// Mitsubishi GX Works2 project: 增压   PLC: FX1S

PROGRAM MAIN
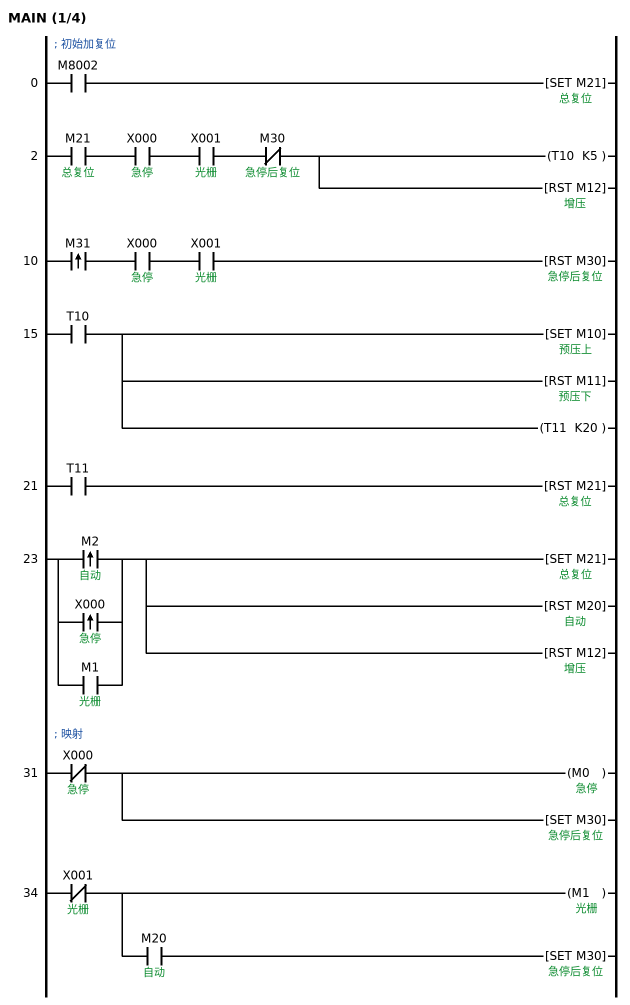
; 初始加复位
0     LD      M8002
      SET     M21  ; 总复位
2     LD      M21  ; 总复位
      AND     X000  ; 急停
      AND     X001  ; 光栅
      ANI     M30  ; 急停后复位
      OUT     T10 K5
      RST     M12  ; 增压
10    LDP     M31
      AND     X000  ; 急停
      AND     X001  ; 光栅
      RST     M30  ; 急停后复位
15    LD      T10
      SET     M10  ; 预压上
      RST     M11  ; 预压下
      OUT     T11 K20
21    LD      T11
      RST     M21  ; 总复位
23    LDP     M2  ; 自动
      ORP     X000  ; 急停
      OR      M1  ; 光栅
      SET     M21  ; 总复位
      RST     M20  ; 自动
      RST     M12  ; 增压
; 映射
31    LDI     X000  ; 急停
      OUT     M0  ; 急停
      SET     M30  ; 急停后复位
34    LDI     X001  ; 光栅
      OUT     M1  ; 光栅
      AND     M20  ; 自动
      SET     M30  ; 急停后复位
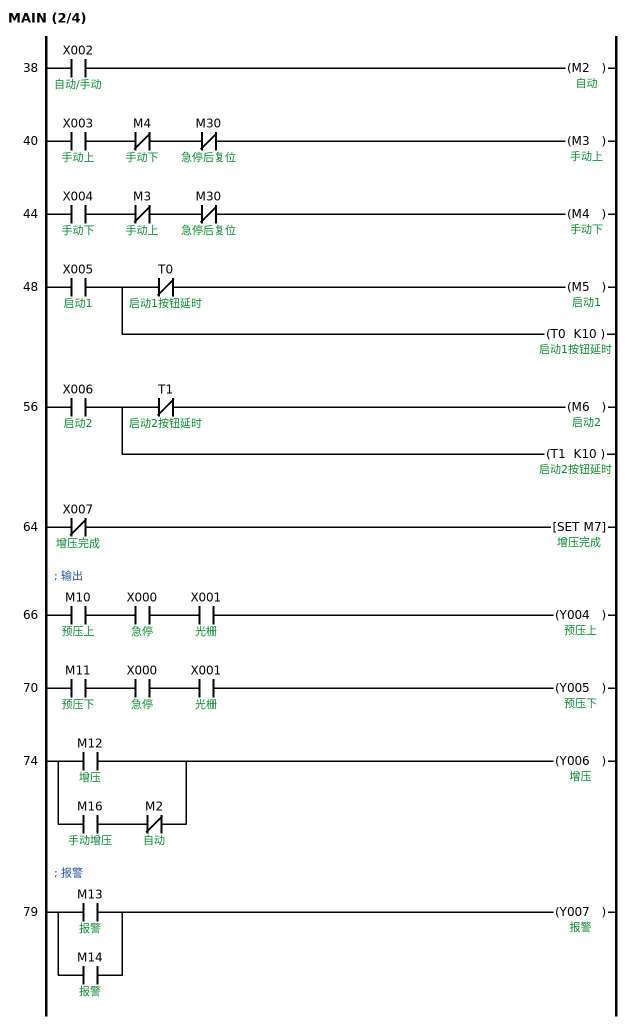
38    LD      X002  ; 自动/手动
      OUT     M2  ; 自动
40    LD      X003  ; 手动上
      ANI     M4  ; 手动下
      ANI     M30  ; 急停后复位
      OUT     M3  ; 手动上
44    LD      X004  ; 手动下
      ANI     M3  ; 手动上
      ANI     M30  ; 急停后复位
      OUT     M4  ; 手动下
48    LD      X005  ; 启动1
      MPS
      ANI     T0  ; 启动1按钮延时
      OUT     M5  ; 启动1
      MPP
      OUT     T0 K10  ; 启动1按钮延时
56    LD      X006  ; 启动2
      MPS
      ANI     T1  ; 启动2按钮延时
      OUT     M6  ; 启动2
      MPP
      OUT     T1 K10  ; 启动2按钮延时
64    LDI     X007  ; 增压完成
      SET     M7  ; 增压完成
; 输出
66    LD      M10  ; 预压上
      AND     X000  ; 急停
      AND     X001  ; 光栅
      OUT     Y004  ; 预压上
70    LD      M11  ; 预压下
      AND     X000  ; 急停
      AND     X001  ; 光栅
      OUT     Y005  ; 预压下
74    LD      M12  ; 增压
      LD      M16  ; 手动增压
      ANI     M2  ; 自动
      ORB
      OUT     Y006  ; 增压
; 报警
79    LD      M13  ; 报警
      OR      M14  ; 报警
      OUT     Y007  ; 报警
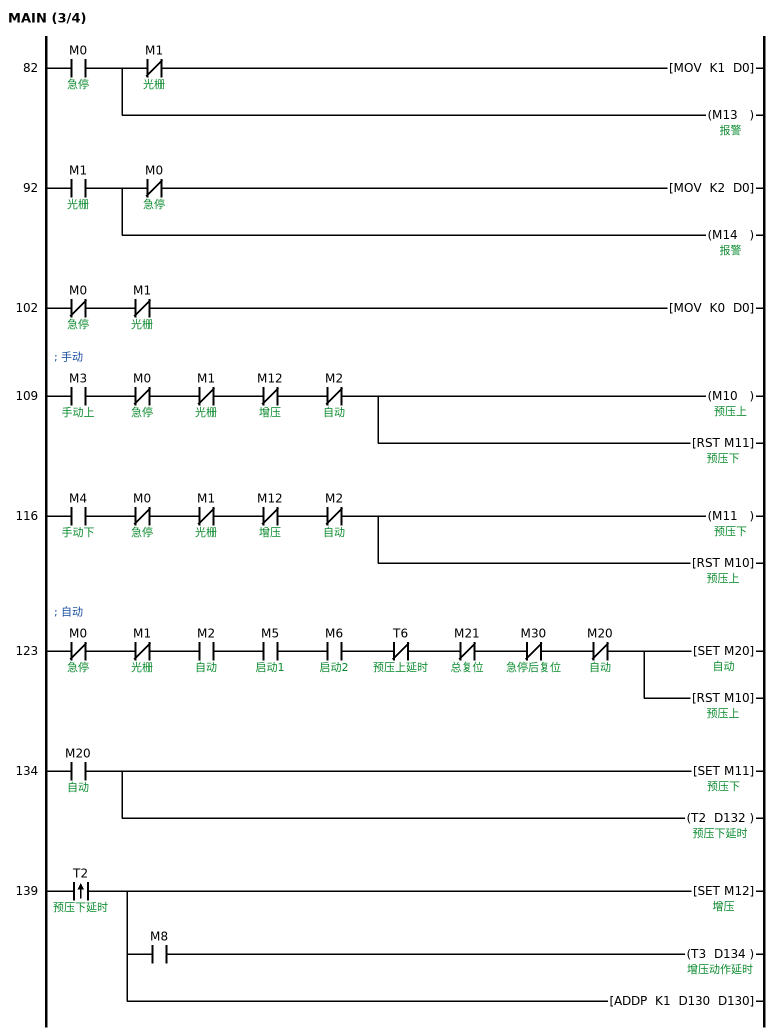
82    LD      M0  ; 急停
      MPS
      ANI     M1  ; 光栅
      MOV     K1 D0
      MPP
      OUT     M13  ; 报警
92    LD      M1  ; 光栅
      MPS
      ANI     M0  ; 急停
      MOV     K2 D0
      MPP
      OUT     M14  ; 报警
102   LDI     M0  ; 急停
      ANI     M1  ; 光栅
      MOV     K0 D0
; 手动
109   LD      M3  ; 手动上
      ANI     M0  ; 急停
      ANI     M1  ; 光栅
      ANI     M12  ; 增压
      ANI     M2  ; 自动
      OUT     M10  ; 预压上
      RST     M11  ; 预压下
116   LD      M4  ; 手动下
      ANI     M0  ; 急停
      ANI     M1  ; 光栅
      ANI     M12  ; 增压
      ANI     M2  ; 自动
      OUT     M11  ; 预压下
      RST     M10  ; 预压上
; 自动
123   LDI     M0  ; 急停
      ANI     M1  ; 光栅
      AND     M2  ; 自动
      AND     M5  ; 启动1
      AND     M6  ; 启动2
      ANI     T6  ; 预压上延时
      ANI     M21  ; 总复位
      ANI     M30  ; 急停后复位
      ANI     M20  ; 自动
      SET     M20  ; 自动
      RST     M10  ; 预压上
134   LD      M20  ; 自动
      SET     M11  ; 预压下
      OUT     T2 D132  ; 预压下延时
139   LDP     T2  ; 预压下延时
      SET     M12  ; 增压
      MPS
      AND     M8
      OUT     T3 D134  ; 增压动作延时
      MPP
      ADDP    K1 D130 D130
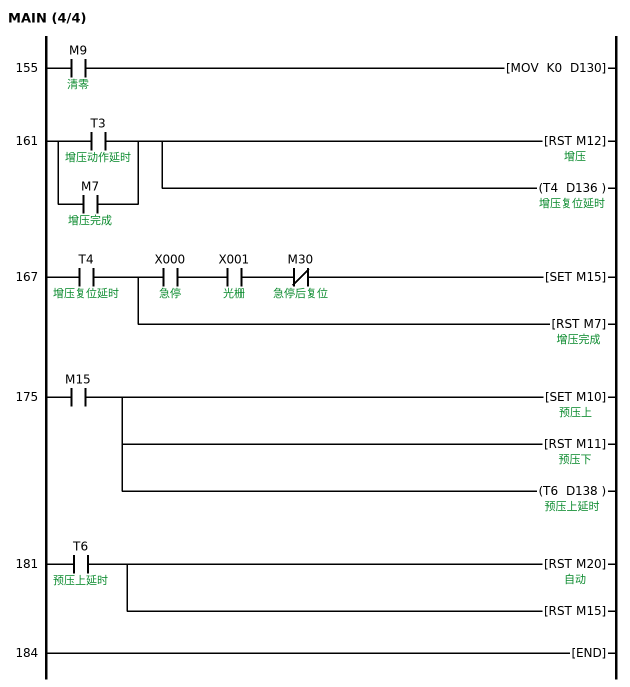
155   LD      M9  ; 清零
      MOV     K0 D130
161   LD      T3  ; 增压动作延时
      OR      M7  ; 增压完成
      RST     M12  ; 增压
      OUT     T4 D136  ; 增压复位延时
167   LD      T4  ; 增压复位延时
      MPS
      AND     X000  ; 急停
      AND     X001  ; 光栅
      ANI     M30  ; 急停后复位
      SET     M15
      MPP
      RST     M7  ; 增压完成
175   LD      M15
      SET     M10  ; 预压上
      RST     M11  ; 预压下
      OUT     T6 D138  ; 预压上延时
181   LD      T6  ; 预压上延时
      RST     M20  ; 自动
      RST     M15
184   END
END_PROGRAM

// device comments not shown above
Y000  ; 预压上
Y001  ; 预压下
Y002  ; 增压
Y003  ; 增压
C0  ; 产量
